INTERFACE PUBLIC LogTargetAdapter EXTENDS __System.IQueryInterface

METHOD PUBLIC Run
END_METHOD

METHOD PUBLIC SendLogEvent : BOOL
VAR_INPUT
	event : LogEvent;
END_VAR
END_METHOD

END_INTERFACE

(* stored: Version 1.1.0.1
   Itf LogTargetAdapter: Id {ac3659bf-3503-42a9-bb64-6b1d9ba4f3f5}
   Method Run: Id {4ddd99af-9e05-4680-8835-ec19bcfc473f}
   Method SendLogEvent: Id {70d2d06d-c23e-42bd-9f71-d1d9247f79db} *)
